Staubli VAL3: goHotel.pgx

program goHotel(num nFrom (dimensions=1))
  local trsf movHorizontal
begin
  //FUTURE ADJUSTMENT: argument nFrom
  //nFrom = 0 -> jHome or pHotel [0] to pHotel[0]
  //nFrom = 1 -> pBeam to pHotel[0]
  switch nFrom
    case 0
      movel(pHotel[0],flange,mNomSpeed)
    break
    case 1
      movel(pBeam,flange,mNomSpeed)
      movel(pHotel2Beam[5],flange,mNomSpeed)
      movel(pHotel2Beam[4],flange,mNomSpeed)
      movel(pHotel2Beam[3],flange,mNomSpeed)
      movel(pHotel2Beam[2],flange,mNomSpeed)
      movel(pHotel2Beam[1],flange,mNomSpeed)
      movel(pHotel2Beam[0],flange,mNomSpeed)
      movel(pHotel[0],flange,mNomSpeed)
    break
    default
      popUpMsg("error goHotel: nFrom"+chr(nFrom))
    break
  endSwitch
  waitEndMove()
end
